{attribute 'linkalways'} 
{attribute 'no_explicit_call' := 'This FB is a CLASS and must be accessed using methods or properties'}
{attribute 'enable_dynamic_creation'}
FUNCTION_BLOCK _ETcVnKnn EXTENDS EnumDatatypeBase
VAR
	localData : ETcVnKnn;
	activeData : REFERENCE TO ETcVnKnn;
	enumBaseDatatype : _UDINT(localData);
END_VAR

METHOD PRIVATE AddLocalEnumeration
VAR_INPUT
	Enumeration : T_MAXSTRING;
	Value : ETcVnKnn;
END_VAR
AddEnumeration(Enumeration, Value);
END_METHOD

PROPERTY PUBLIC Address : PVOID
GET
Address := ADR(activeData);
END_GET
END_PROPERTY

METHOD PUBLIC ClearReference
VAR_INPUT
END_VAR
activeData REF= localData;
SetBaseDatatypeReference();
END_METHOD

METHOD PUBLIC Clone : I_Datatype
VAR
    pClone : POINTER TO _ETcVnKnn;
END_VAR
pClone := __NEW(_ETcVnKnn(InitialValue := Value));
Clone := pClone^;
END_METHOD

METHOD FB_init : BOOL
VAR_INPUT
	bInitRetains : BOOL; // if TRUE, the retain variables are initialized (warm start / cold start)
	bInCopyCode : BOOL;  // if TRUE, the instance afterwards gets moved into the copy code (online change)
	InitialValue : ETcVnKnn;
END_VAR
localData := InitialValue;
AddBaseDatatype(enumBaseDatatype);
ClearReference();

AddLocalEnumeration('TCVN_KNN_CLASSIFIER', ETcVnKnn.TCVN_KNN_CLASSIFIER);
AddLocalEnumeration('TCVN_KNN_NOVELTY_DETECTOR', ETcVnKnn.TCVN_KNN_NOVELTY_DETECTOR);
AddLocalEnumeration('TCVN_KNN_REGRESSOR', ETcVnKnn.TCVN_KNN_REGRESSOR);
END_METHOD

PROPERTY PUBLIC Identifier : T_MAXSTRING
GET
Identifier := 'ETcVnKnn';
END_GET
END_PROPERTY

METHOD IsEnumeratorValueEqual : BOOL
VAR_INPUT
	Enumerator : I_KeyValueForwardEnumerator;
END_VAR
VAR
	storedValue : ETcVnKnn;
END_VAR
IF NOT Enumerator.TryGet(storedValue) THEN
	RETURN;
END_IF

IsEnumeratorValueEqual := storedValue = activeData;
END_METHOD

METHOD PUBLIC MakeReferenceTo
VAR_INPUT
	ReferenceTarget : REFERENCE TO ETcVnKnn;
END_VAR
activeData REF= ReferenceTarget;
SetBaseDatatypeReference();
END_METHOD

METHOD PROTECTED SetBaseDatatypeReference
VAR_INPUT
END_VAR
enumBaseDatatype.MakeReferenceTo(activeData);
END_METHOD

PROPERTY PUBLIC Size : UDINT
GET
Size := SIZEOF(activeData);
END_GET
END_PROPERTY

METHOD TryMakeReferenceTo : BOOL
VAR_INPUT
	Target : I_Datatype;
END_VAR
VAR
	targetAsEnum : I_EnumDatatype;
	pTargetData : POINTER TO ETcVnKnn;
END_VAR
IF NOT Target.TryResolveAsEnumDatatype(targetAsEnum) THEN
	RETURN;
END_IF

IF targetAsEnum.Identifier <> Identifier THEN
	RETURN;
END_IF

pTargetData := Target.Address;
activeData REF= pTargetData^;
SetBaseDatatypeReference();
TryMakeReferenceTo := TRUE;
END_METHOD

PROPERTY PUBLIC Value : ETcVnKnn
GET
Value := activeData;
END_GET
SET
activeData := Value;
END_SET
END_PROPERTY

END_FUNCTION_BLOCK

(* stored: Version 1.1.0.1, ProductVersion 3.1.4024.12
   POU _ETcVnKnn: Id {d4c160ab-c5ca-4c57-84bd-9079faf054a2}, SpecialFunc None
   Folder Constructor: Id {8fc76e67-b17c-4a5a-96a8-456e0538ea31}
   Folder Private: Id {8f1437f5-ccac-4acd-90fa-54d33bb91a70}
   Folder Protected: Id {97e3aa03-65a9-4bcb-a735-dab7cb5c75f9}
   Method AddLocalEnumeration: Id {f36d0f49-0abc-498e-8b35-e87357ed2523}
   Property Address: Id {cf2f3eea-102b-4bb4-9077-37482ad06c4c}
   Get Get: Id {28784cb6-4d23-4631-83fc-6f73f51158d7}
   Method ClearReference: Id {a9c5d1e7-8160-45cd-b6f1-cd427babd1b7}
   Method Clone: Id {6a36dfa1-4406-4c24-9c0e-ca52e4358c8d}
   Method FB_init: Id {16ef6e1b-740e-4d71-bdf3-c4d4b75852b1}
   Property Identifier: Id {252a4266-ad53-42b6-9214-0cafc84c009a}
   Get Get: Id {900242d1-141f-4c78-a915-3f8f546129ae}
   Method IsEnumeratorValueEqual: Id {227696f3-1b00-4a15-b28c-403630ba9aad}
   Method MakeReferenceTo: Id {f1d4af9a-ef3f-4f39-b08f-1119060bc6ec}
   Method SetBaseDatatypeReference: Id {02b9b3bf-ec25-4962-a56d-559d2f613f9b}
   Property Size: Id {3200956f-e740-4453-86db-06196bd59e8d}
   Get Get: Id {019d44b5-6378-46db-b818-fce4679d4daf}
   Method TryMakeReferenceTo: Id {7bfed5fd-7935-452d-add1-17a1004e552c}
   Property Value: Id {120b28ae-a9bf-44ca-803a-f00235ac69f4}
   Get Get: Id {2e18971f-0572-4fef-89bf-9df5c2f00d75}
   Set Set: Id {fda23341-05b1-494c-96ac-56533dbacf7e} *)
